TYPE MultipleEventTestsystem :
STRUCT
  runner: EventRunner;
  event1: Event := (runner:=runner);
  event2: Event := (runner:=runner);
  event3: Event := (runner:=runner);
END_STRUCT
END_TYPE

(* stored: Version 1.1.0.1, ProductVersion 3.1.4024.9
   DUT MultipleEventTestsystem: Id {463db442-f089-4be4-9631-f04acbc95b47} *)
